TYPE ST_IOOutputSimul :
STRUCT
	QxLampeRouge AT%Q*:BOOL;
END_STRUCT
END_TYPE

(* stored: Version 1.1.0.1, ProductVersion 3.1.4020.6
   DUT ST_IOOutputSimul: Id {8ef0b6d5-238d-47ba-a7f5-b954781fe0a8} *)
